// TIA Portal V20 export
DATA_BLOCK "BK18"   // DB264
// stored: MemoryReserve 100
   VAR
      "X10-1 WEIGHT NG CLAMP MOVER OPEN" : Bool;
      "X11-1 WEIGHT NG CLAMP LEFT OPEN" : Bool;
      "X12-1 WEIGHT NG CLAMP RIGHT OPEN" : Bool;
      "X13-1 WEIGHT NG CLAMP Z-AXIS UP" : Bool;
      "X14-1 WEIGHT NG CLAMP MOVER BACKWARD" : Bool;
      "X15-1 WEIGHT NG BOX LIFT DOWN" : Bool;
      "X16-1 WEIGHT NG BOX LOCK DOWN" : Bool;
      "X17-1 STACK NG FULL SENSOR" : Bool;
      "X10-2 WEIGHT NG CLAMP MOVER CLOSE" : Bool;
      "X11-2 WEIGHT NG CLAMP LEFT CLOSE" : Bool;
      "X12-2 WEIGHT NG CLAMP RIGHT CLOSE" : Bool;
      "X13-2 WEIGHT NG CLAMP Z-AXIS DOWN" : Bool;
      "X14-2 WEIGHT NG CLAMP MOVER FORWARD" : Bool;
      "X15-2 WEIGHT NG BOX LIFT UP" : Bool;
      "X16-2 WEIGHT NG BOX LOCK UP" : Bool;
      "X17-2 SPARE" : Bool;
   END_VAR
BEGIN
END_DATA_BLOCK
